FUNCTION_BLOCK ExampleFB (* Example Function Block *)
  (* Version 1.0, 2024-01-01, Test *)
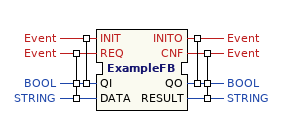
  EVENT_INPUT
    INIT WITH QI; (* Initialization *)
    REQ WITH QI, DATA; (* Request *)
  END_EVENT
  EVENT_OUTPUT
    INITO WITH QO; (* Initialization Confirm *)
    CNF WITH QO, RESULT; (* Confirmation *)
  END_EVENT
  VAR_INPUT
    QI : BOOL; (* Qualifier Input *)
    DATA : STRING; (* Input Data *)
  END_VAR
  VAR_OUTPUT
    QO : BOOL; (* Qualifier Output *)
    RESULT : STRING; (* Result Data *)
  END_VAR
END_FUNCTION_BLOCK
